PROGRAM PRG_COM
VAR
END_VAR

//needs to run on a seperate task

(*Instanitate Serial port com function *)
//LXLHN_PTM_01
PTM_fbSerialLineControl(
	Mode:= SERIALLINEMODE_EL6_22B,
	pComIn:= ADR(PTM_stComIn),
	pComOut:=ADR(PTM_stComOut),
	SizeComIn:= SIZEOF(PTM_stComOut),
	TxBuffer:= PTM_SerialTXBuffer,
	RxBuffer:= PTM_SerialRXBuffer,
	Error=> ,
	ErrorID=> );

END_PROGRAM

(* stored: Version 1.1.0.1, ProductVersion 3.1.4022.18
   POU PRG_COM: Id {b34d4e82-5727-4a29-885a-665d0a9d3503}, SpecialFunc None *)
